{attribute addProperty BoxType "EL2911-0000-0016"}
{attribute addProperty Id "FSoE_InputsFSoE_Inputs_1D066A9C486FSoE_OutputsFSoE_Outputs_6FE7597C486"}
{attribute addProperty CRC "1640139511"}
{attribute addProperty SizeInBites "96"}
{attribute addProperty SizeInBytes "12"}
TYPE Module_1_FSOE_61C28AF7 :
STRUCT
	{attribute addProperty Name "FSoE_Inputs"}
	FSoE_Inputs  : FSoE_Inputs_1D066A9C;
	{attribute addProperty Name "FSoE_Outputs"}
	FSoE_Outputs  : FSoE_Outputs_6FE7597C;
END_STRUCT
END_TYPE

(* stored: Version 1.2.0.0, ProductVersion 3.1.4024.9
   DUT Module_1_FSOE_61C28AF7: Id {fa19a4df-4660-4595-961b-8d06682c5e38} *)
